FUNCTION_BLOCK FB_Alarm
VAR
	_usedCore 			: IAlarmCore;
END_VAR
VAR_STAT
  	_coreSingletonInstance : IAlarmCore;
END_VAR

METHOD PRIVATE Initialize : BOOL
VAR_INPUT
END_VAR
IF (_usedCore = 0) THEN 
	_usedCore := _coreSingletonInstance; 
END_IF
END_METHOD

METHOD RaiseAlarm
VAR_INPUT
	alarmMessage : STRING;
END_VAR
Initialize();
_usedCore.AddAlarm(alarmMessage);
END_METHOD

METHOD SetCore : BOOL
VAR_INPUT
  	ref2Core : IAlarmCore; 
END_VAR
_coreSingletonInstance := ref2Core;
END_METHOD

END_FUNCTION_BLOCK

(* stored: Version 1.1.0.1, ProductVersion 3.1.4024.12
   POU FB_Alarm: Id {a16a4457-e980-4d70-9b79-85bb55c618bc}, SpecialFunc None
   Method Initialize: Id {2c7319f7-5db0-41d0-a3f2-cc4525239a30}
   Method RaiseAlarm: Id {f90c2a31-76b6-4bf1-a3c6-48cfa816c3ef}
   Method SetCore: Id {e39d7376-bcf9-45e8-a074-b4fff7d687e5} *)
